// Mitsubishi GX Works2 project: Manual forward reverse   PLC: FX1S

PROGRAM MAIN
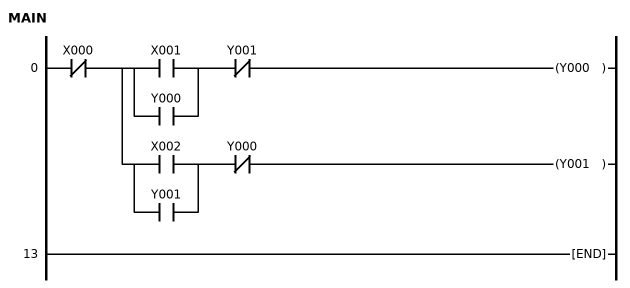
0     LDI     X000
      MPS
      LD      X001
      OR      Y000
      ANB
      ANI     Y001
      OUT     Y000
      MPP
      LD      X002
      OR      Y001
      ANB
      ANI     Y000
      OUT     Y001
13    END
END_PROGRAM
